// TIA Portal V19 export
DATA_BLOCK "AUTO_SUBOUTPUT DB"   // DB58
{ S7_Optimized_Access := 'TRUE' }
// stored: MemoryReserve 100
   VAR
      "MGF FEED PUMP P-101 A" : Bool;
      "MGF FEED PUMP P-101 B" : Bool;
      "MGF BACK WASH P-102 A" : Bool;
      "MGF BACK WASH P-102 B" : Bool;
      "UF FEED PUMP P-103 A" : Bool;
      "UF FEED PUMP P-103 B" : Bool;
      "UF BLOWER AB-201 A" : Bool;
      "UF BLOWER AB 201 B" : Bool;
      "UF BACK WASH P-201 A" : Bool;
      "UF BACK WASH  P-201 B" : Bool;
      "DM FEED PUMP P-502 A" : Bool;
      "DM FEED PUMP P-502 B" : Bool;
      "DM FEED PUMP P-502 C" : Bool;
      "CIP PUMP P-601" : Bool;
      "BACK WASH RECOVERY P-801 A" : Bool;
      "BACK WASH RECOVERY P-801 B" : Bool;
      SPARE : Bool;
      "SPARE(1)" : Bool;
      "SPARE(2)" : Bool;
      "DP-701" : Bool;
      "DP-702" : Bool;
      "NaOCL DOSING D-706 A" : Bool;
      "NaOCL DOSING DP-706B" : Bool;
      "ABFV-501" : Bool;
      "ABFV-502" : Bool;
      "ABFV 101 MULTIGRADE FILTER VALVE" : Bool;
      "ABFV 102 MULTIGRADE FILTER VALVE" : Bool;
      "ABFV 103 MULTIGRADE FILTER VALVE" : Bool;
      "ABFV 104 MULTIGRADE FILTER VALVE" : Bool;
      "ABFV 105 MULTIGRADE FILTER VALVE" : Bool;
      "ABV 201 UF VALVE" : Bool;
      "ABFV 201 UF VALVE" : Bool;
      "ABFV 202 UF VALVE" : Bool;
      "ABFV 203 UF VALVE" : Bool;
      "ABFV 204 UF VALVE" : Bool;
      "ABFV 205 UF VALVE" : Bool;
      "ABFV 206 UF VALVE" : Bool;
      "ABFV 207 UF VALVE" : Bool;
      "ABFV 208 UF VALVE" : Bool;
   END_VAR
BEGIN
END_DATA_BLOCK
